TYPE RampConfiguration EXTENDS BaseConfiguration:
STRUCT
END_STRUCT
END_TYPE

(* stored: Version 1.1.0.1
   DUT RampConfiguration: Id {8a582694-8d2b-4d37-aa92-6e6f09e5e984} *)
